FUNCTION_BLOCK MoveAbs IMPLEMENTS I_MoveAbs
VAR
	mcMoveAbs : MC_MoveAbsolute;
END_VAR
VAR_IN_OUT
	Axis : AXIS_REF;
END_VAR

mcMoveAbs(Axis := Axis);

PROPERTY Acceleration : MC_LREAL
GET
Acceleration := mcMoveAbs.Acceleration;
END_GET
SET
mcMoveAbs.Acceleration := Acceleration;
END_SET
END_PROPERTY

PROPERTY BufferMode : MC_Buffermode
GET
BufferMode := mcMoveAbs.BufferMode;
END_GET
SET
mcMoveAbs.BufferMode := BufferMode;
END_SET
END_PROPERTY

PROPERTY Busy : BOOL
GET
Busy := mcMoveAbs.Busy;
END_GET
END_PROPERTY

PROPERTY Deceleration : MC_LREAL
GET
Deceleration := mcMoveAbs.Deceleration;
END_GET
SET
mcMoveAbs.Deceleration := Deceleration;
END_SET
END_PROPERTY

PROPERTY Done : BOOL
GET
Done := mcMoveAbs.Done;
END_GET
END_PROPERTY

PROPERTY Error : BOOL
GET
Error := mcMoveAbs.Error;
END_GET
END_PROPERTY

PROPERTY Execute : BOOL
GET
Execute := mcMoveAbs.Execute;
END_GET
SET
mcMoveAbs.Execute := Execute;
END_SET
END_PROPERTY

PROPERTY Jerk : MC_LREAL
GET
Jerk := mcMoveAbs.Jerk;
END_GET
SET
mcMoveAbs.Jerk := Jerk;
END_SET
END_PROPERTY

PROPERTY Position : MC_LREAL
GET
Position := mcMoveAbs.Position;
END_GET
SET
mcMoveAbs.Position := Position;
END_SET
END_PROPERTY

PROPERTY Velocity : MC_LREAL
GET
Velocity := mcMoveAbs.Velocity;
END_GET
SET
mcMoveAbs.Velocity := Velocity;
END_SET
END_PROPERTY

END_FUNCTION_BLOCK

(* stored: Version 1.1.0.1
   POU MoveAbs: Id {2564abcd-200b-46fd-8045-7789bc59a486}, SpecialFunc None
   Property Acceleration: Id {b95cd058-3a55-4e61-870f-cc7e2c69546d}
   Get Get: Id {575c6061-1e40-43fc-84d3-0a827e349f5b}
   Set Set: Id {338c95cb-d15f-44aa-93f0-ecedfbc0d6fd}
   Property BufferMode: Id {12974983-43d9-4de1-874c-c9269d5878c1}
   Get Get: Id {8d8815da-9ec9-4748-bbdc-d84333d8b33e}
   Set Set: Id {b307df7c-cc0e-48b0-bac0-e52cfed79467}
   Property Busy: Id {60a1567b-b733-46b5-b4bc-4e0bfe590134}
   Get Get: Id {e72e88fa-1b6d-4214-beab-e34e2fcfa155}
   Property Deceleration: Id {552ca7c4-5eb6-4638-aa1c-b9a1815723c6}
   Get Get: Id {a518ffc4-a923-4b9f-af82-f28f668dc357}
   Set Set: Id {e50bdb2b-7008-4235-85dc-bac731a513ed}
   Property Done: Id {3b499f05-39a4-4dc2-be56-124c5716b051}
   Get Get: Id {eb4de39c-12b4-4990-9ed4-66be250d3f38}
   Property Error: Id {280506ff-d6b7-4352-982e-5f2801de4ea6}
   Get Get: Id {9ab70db9-3b74-493e-8c58-c8d3d310abf7}
   Property Execute: Id {80fb8c86-89fe-4d60-85b8-183273bfef7a}
   Get Get: Id {bb39a42b-d0d3-401c-a8a4-e1bad5de7647}
   Set Set: Id {2926150f-7f00-4170-87ec-408ddda0c8c7}
   Property Jerk: Id {19a58d80-740d-4fa6-9d27-944abf5123d2}
   Get Get: Id {4505ab81-f2d9-41b1-978e-89ed106f3fd0}
   Set Set: Id {0456f2ac-7215-47d1-9cc5-08fdbaa3540b}
   Property Position: Id {071894e5-07d8-4e43-948b-52a14e523eed}
   Get Get: Id {b3a2faca-7b49-459d-a548-f5ab5c7230cd}
   Set Set: Id {a35a343f-c1e4-4e06-8023-2c9078efbf29}
   Property Velocity: Id {41a2c790-a30a-425f-b898-da47debd5503}
   Get Get: Id {355a2ac1-3405-425f-b36a-1e3c8ea1dce7}
   Set Set: Id {65d6d285-747e-4fb9-867e-b621d1184a9f} *)
